// SIMATIC S7-200 project (STEP 7-Micro/WIN), CPU 221 REL 01.10

ORGANIZATION_BLOCK 主程序:OB1
TITLE=程序注释
BEGIN
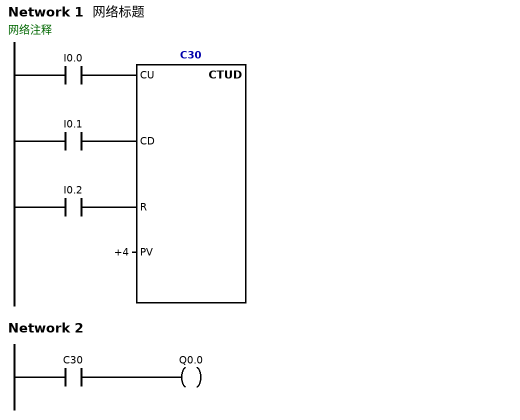
Network 1 // 网络标题
// 网络注释
// (network saved uncompiled; LAD cells follow)
// row 0: c0 -| |- I0.0  c1 [CTUD C30 CU:=power@row0, CD:=power@row1, R:=power@row2, PV:=+4]
// row 1: c0 -| |- I0.1  c1 [box]
// row 2: c0 -| |- I0.2  c1 [box]
// row 3: c1 [box]
Network 2
// (network saved uncompiled; LAD cells follow)
// row 0: c0 -| |- C30  c1 -( ) Q0.0
END_ORGANIZATION_BLOCK
